RoboDK station: DynamicTarget.rdk

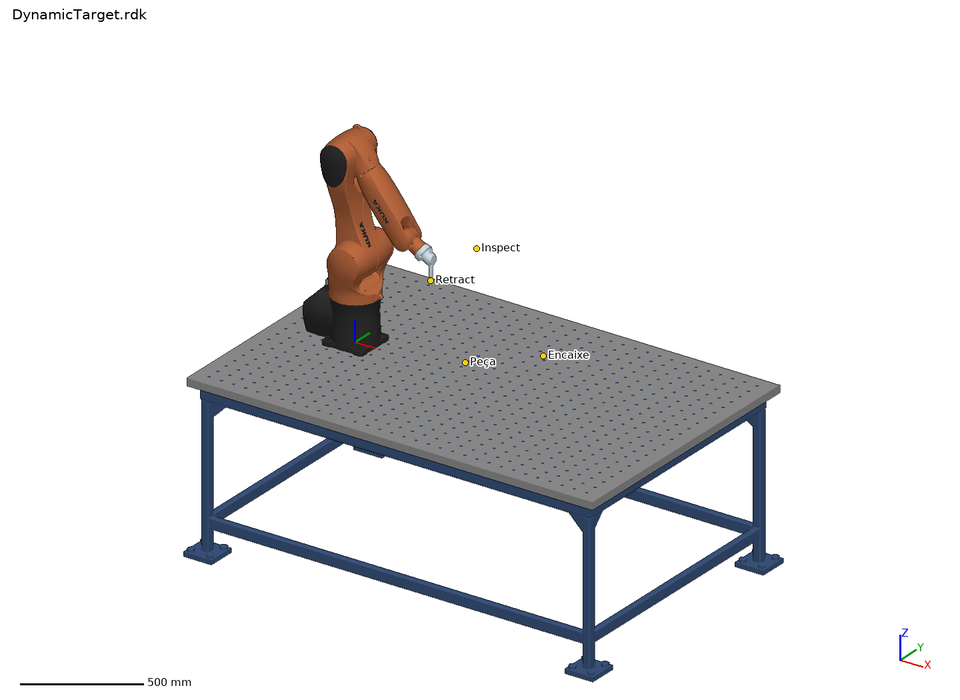
[picture v0: the station drawn from its stored meshes, robots at their saved joint values, targets as dots, program paths as lines]
Station DynamicTarget (saved by RoboDK 5.5.2). Poses are relative to the parent item; angles as X-Y-Z fixed-axis rotations.
  - frame Base at (-207.87, 0, -62.35) mm
    - robot Robot (model KUKA KR 6 R900 sixx): 6 axes, payload 6 kg, reach 901 mm, repeatability 0.03 mm, weight 52 kg
        modified DH rows (alpha deg, a mm, theta deg, d mm): 0, 0, 0, 400; -90, 25, 0, 0; 0, 455, -90, 0; -90, 35, 0, 420; 90, 0, 0, 0; -90, 0, 180, 80
        joint limits [-170, -190, -120, -185, -120, -350] to [170, 45, 156, 185, 120, 350]; home [0, -90, 90, 0, 0, 0]; saved at [-0.563, -97.056, 149.262, 178.71, 22.21, -179.087]
      - tool Pencil, TCP at (82.2, 0, 101.78) mm, rotated rx 0 ry 60 rz 0 deg, size 74.9 x 125 x 107.3 mm
    - target Inspect (Cartesian target) at (595.41, 2.5, 584.69) mm, rotated rx 180 ry 0 rz -180 deg; joints [-0.299, -84.178, 103.493, 181.395, -10.689, -181.52] of Robot
    - target Retract (Cartesian target) at (370.47, 2.5, 379.03) mm, rotated rx 180 ry 0 rz -180 deg; joints [-0.563, -97.056, 149.262, 178.71, 22.21, -179.087] of Robot
    - object Table at (0, 0, 0) mm, size 2020 x 1340 x 800 mm, geometry from Table-2000x1200x800mm.sld
    - target Peça (Cartesian target) at (473, 101, 0) mm, rotated rx -180 ry 0 rz -180 deg; joints [-101.614, 14.834, 153.184, 118.098, 74.077, -265.148] of Robot
    - target Encaixe (Cartesian target) at (695, 331, 0) mm, rotated rx -180 ry 0 rz -180 deg; joints [-101.614, 14.834, 153.184, 118.098, 74.077, -265.148] of Robot
  - Python program dynamicTarget (listed below)

--- Python program dynamicTarget ---
from robodk.robolink import *      # RoboDK's API
from robodk.robomath import *      # Math toolbox for robots
from tkinter import *
import numpy as np
import cv2

def getElements(image):
    imgHSV = cv2.cvtColor(image, cv2.COLOR_BGR2HSV)
    lower = np.array([32, 0, 0])
    upper = np.array([145, 255, 255])
    mask = cv2.inRange(imgHSV, lower, upper)
    imgResult = cv2.bitwise_and(image, image, mask=mask)
    return imgResult

def showImages(images):
    for image in images:
        cv2.imshow('Image', image)
        cv2.waitKey(0)
        cv2.destroyAllWindows()

def getPosition():
    path = 'C:/Code/IC-Gemeo-master/IC-Gemeo-master/Localizacao de Objetos/Exemplo/bancada1.png'
    image = cv2.imread(path)
    #image = cv2.resize(image, (1200, 2000))
    maskedImage = getElements(image)

    img = maskedImage.copy()
    im_bw = cv2.cvtColor(img, cv2.COLOR_RGB2GRAY)
    #blur = cv2.GaussianBlur(im_bw, (5,5), 0)
    #im_bw = cv2.Canny(blur, 10, 90)
    contours, hierarchy = cv2.findContours(im_bw, cv2.RETR_TREE, cv2.CHAIN_APPROX_SIMPLE)
    centers = []
    for c in contours:
        M = cv2.moments(c)
        if M['m00'] != 0:
            cx = int(M['m10']/M['m00'])
            cy = int(M['m01']/M['m00'])
            cv2.drawContours(img, [c], -1, (0,255,0), 3)
            cv2.circle(img, (cx, cy), 5, (0,0,255), -1)
            cv2.putText(img, f"{cx, cy}", (cx - 20, cy - 20), cv2.FONT_HERSHEY_SIMPLEX, 0.5, (0,0,255), 2)
            centers.append((cx, cy))
    showImages([image, maskedImage, img])
    return centers

def interface():
    centers = getPosition()

    master = Tk()
    master.geometry("400x400")
    master.title("Localização de Objetos")
    master.eval('tk::PlaceWindow . center')


    t = Text(master, height=10, width=10)
    for x in centers:
        t.insert(END, x)
        t.insert(END, "\n")
    t.pack()

    indexes = []
    j = 0
    for _ in centers:
        indexes.append(j)
        j += 1

    variable = StringVar(master)
    variable.set(indexes[0])

    w = OptionMenu(master, variable, *indexes)
    w.pack()


    def ok():
        result = variable.get()
        print ("value is: " + result)
        print(centers[int(result)])
        global cx, cy
        cx, cy = centers[int(result)]
        master.destroy()

    button = Button(master, text="OK", command=ok)
    button.pack()

    mainloop()
    return cx, cy

RL = Robolink()

robot = RL.Item('Robot')
base = RL.Item('Base')
inspect = RL.Item('Inspect')
retract = RL.Item('Retract')

target = RL.AddTarget('Cube', base)
cx, cy = interface()
print(cx, cy)
RL.ShowMessage('Centers: ' + str(cx) + ' ' + str(cy))
target.setPose(Offset(eye(), cx, cy, 0, -180, 0, 180))

robot.MoveJ(inspect)
robot.MoveJ(target)
robot.MoveJ(retract)
